PROGRAM ModeManger
VAR
END_VAR

IF GVL_Machine.ModeUI = 'Auto' THEN 
	GVL_Machine.machineMode := MachineMode.Auto;
ELSIF GVL_Machine.ModeUI = 'Manual' THEN 
	GVL_Machine.machineMode := MachineMode.Manual;	
ELSIF	GVL_Machine.ModeUI ='Setting' THEN 
	GVL_Machine.machineMode := MachineMode.Setting;
ELSIF GVL_Machine.ModeUI = 'Calibration' THEN 
	GVL_Machine.machineMode := MachineMode.Calibration;
ELSE
	GVL_Machine.machineMode := MachineMode.Idle;
END_IF


//transer the machine mode to PLC Main page
CASE GVL_Machine.machineMode OF
	MachineMode.Auto:
		GVL_Machine.ModePLC := 'Auto';
	MachineMode.Manual:
		GVL_Machine.ModePLC := 'Manual';	
	MachineMode.Idle:
		GVL_Machine.ModePLC := 'Idle';
	MachineMode.Calibration:
		GVL_Machine.ModePLC := 'Calibration';
	MachineMode.Setting:
		GVL_Machine.ModePLC := 'Setting';
	MachineMode.Undefined:
		GVL_Machine.ModePLC := 'Undefined';	
END_CASE

END_PROGRAM

(* stored: Version 1.1.0.1, ProductVersion 3.1.4022.16
   POU ModeManger: Id {c86caeba-dcb1-4820-a4b8-dc420e7c71f2}, SpecialFunc None *)
